// TIA Portal V20 export
// export: Created 2025-12-01T14:56:21.8994682Z, ExportSetting None, DisplayName Totally Integrated Automation Portal, DisplayVersion V20 Update 3, DisplayName TIA Portal Openness, DisplayVersion V20 Update 3, DisplayName TIA Portal Version Control Interface, DisplayVersion V20 Update 3, DisplayName STEP 7 Professional, DisplayVersion V20 Update 3, DisplayName STEP 7 Safety, DisplayVersion V20 Update 2, DisplayName WinCC Basic/Comfort/Advanced, DisplayVersion V20 Update 3, DisplayName WinCC Professional, DisplayVersion V20 Update 3, DisplayName WinCC Unified, DisplayVersion V20 Update 3
TYPE "CBS_Elemento"
   STRUCT
      posicion_real_elemento : Real;   // Posición que ocupa el elemento medido en mm desde el punto 0 del sistema
      ventana_minima : Int;   // Valor minimo de avance para considerar que el vagón se encuentra en ventana
      ventana_maxima : Int;   // Valor máximo de avance para considerar que el vagón se encuentra en ventana
      ID_Destino_Derecha : Int;
      ID_Destino_Izquierda : Int;
      Hay_Carrier_en_ventana : Bool;   // Indica que el vagón se encuentra dentro de la ventana del elemento
      Reserva_1 : Bool;   // Reserva
      Reserva_2 : Bool;   // Reserva
      Reserva_3 : Bool;   // Reserva
      Reserva_4 : Bool;   // Reserva
      Reserva_5 : Bool;   // Reserva
      Reserva_6 : Bool;   // Reserva
      Reserva_7 : Bool;   // Reserva
      Numero_carrier : Int;   // Vagon que se encuentra frente al elemento.
      Avance_carrier : Int;   // Distancia que sobrepasa el vagon la posición del elemento en mm.
   END_STRUCT;
END_TYPE
